FUNCTION_BLOCK E_SPLIT_4 (* Split an event (generic FB) *)
  {SET_ATTRIBUTE(eclipse4diac::core::GenericClassName, 'GEN_E_SPLIT')}
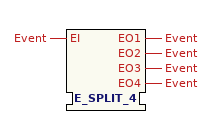
  EVENT_INPUT
    EI; (* Input event *)
  END_EVENT
  EVENT_OUTPUT
    EO1; (* First output event *)
    EO2; (* Second output event *)
    EO3;
    EO4;
  END_EVENT
END_FUNCTION_BLOCK
